Fanuc KAREL source: kt00493.KL

-- PROVISIONAL review KL for V940-1; original PC SHA256 2e21c41f844630f253cc1474472e26cf50779b9ad701b3209c3860c7e2ef0967
-- Incomplete behavior may be omitted. Consult companion uncertainty JSON. Do not deploy.
PROGRAM KT00493
%NOLOCKGROUP
VAR
  OUT : BOOLEAN
-- UNRESOLVED_DECL P1 type=000102
-- UNRESOLVED_DECL P2 type=000101
BEGIN
  -- V9_ZERO_TABLE_METADATA_HINT layout=0001; no indexed target words; source/name/runtime held
  -- UNRESOLVED_PC offsets 5-20; opcodes 2E,22,32,35
  -- UNRESOLVED_PC offsets 25-53; opcodes 49,7E,49,AC,23
  -- UNRESOLVED_PC offsets 58-62; opcodes 7F
END KT00493
